// TIA Portal V19 export
TYPE "LAF_typeSequenceStatus"
// Status of the sequence
// stored: Access Published
   STRUCT
      automaticMode { ExternalWritable := 'False'} : Bool;   // In Automatic Mode
      singleStepMode { ExternalWritable := 'False'} : Bool;   // In Single Step Mode
      currentStep { ExternalWritable := 'False'} : DInt;   // Current step
      nextStep { ExternalWritable := 'False'} : DInt;   // Next selected step
      previousStep { ExternalWritable := 'False'} : DInt;   // Step before current step
      currentStepSTRING { ExternalWritable := 'False'} : String;   // Current step
      nextStepSTRING { ExternalWritable := 'False'} : String;   // Next selected step
      previousStepSTRING { ExternalWritable := 'False'} : String;   // Step before current step
      inStepIdle { ExternalWritable := 'False'} : Bool;   // Sequence in step IDLE
      inStepStopped { ExternalWritable := 'False'} : Bool;   // Sequence in step STOPPED
      seqActive { ExternalWritable := 'False'} : Bool;   // Sequence active
      stepActive { ExternalWritable := 'False'} : Bool;   // Current step is active
      stepComplete { ExternalWritable := 'False'} : Bool;   // Currently active step is complete
      executionEnabled { ExternalWritable := 'False'} : Bool;   // Execution is enabled, move from idle to first process step
      initRequired { ExternalWritable := 'False'} : Bool;   // Init commands requested to continue
      stepChangeReleased { ExternalWritable := 'False'} : Bool;   // Jumping to next step is released
      justSteppedPulse { ExternalWritable := 'False'} : Bool;   // Just changed the step
      manualControlEnabled { ExternalWritable := 'False'} : Bool;   // Control via moduleInterface enabled
      manualModeChangeEnabled { ExternalWritable := 'False'} : Bool;   // Manual mode change possible (only if manualControl is enabled)
      memoryStepTimer { ExternalWritable := 'False'} : LReal;   // Internal bit to memorize time of step entry
   END_STRUCT;
END_TYPE
